Fanuc KAREL source: CA0046.KL

PROGRAM CA0046
%STACKSIZE=65535
%PRIORITY=65535
%NOLOCKGROUP
TYPE
T=STRUCTURE
A : INTEGER
B : REAL
ENDSTRUCTURE
VAR
G : INTEGER
I : INTEGER
R : REAL
B : BOOLEAN
S : STRING[16]
AI : ARRAY[2] OF INTEGER
AR : ARRAY[2] OF REAL
ST : T
P : XYZWPR
V : VECTOR
ROUTINE F(P1 : ARRAY[*] OF INTEGER; P2 : ARRAY[*] OF REAL; P3 : T; P4 : XYZWPR; P5 : VECTOR; P6 : ARRAY[*] OF INTEGER; P7 : ARRAY[*] OF REAL; P8 : T; P9 : XYZWPR; P10 : VECTOR; P11 : ARRAY[*] OF INTEGER;
P12 : ARRAY[*] OF REAL; P13 : T; P14 : XYZWPR; P15 : VECTOR; P16 : ARRAY[*] OF INTEGER; P17 : ARRAY[*] OF REAL; P18 : T; P19 : XYZWPR; P20 : VECTOR; P21 : ARRAY[*] OF INTEGER; P22 : ARRAY[*] OF REAL;
P23 : T; P24 : XYZWPR) FROM CA0046
ROUTINE F
BEGIN
G=(G + 1)
END F
BEGIN
G=0
I=1
R=2.5
B=TRUE
S='A'
AI[1]=3
AR[1]=4.5
-- UNSAFE_SOURCE_IR line 54: ST.A = 5
-- UNSAFE_SOURCE_IR line 55: ST.B = 6.5
F(AI,AR,ST,P,V,AI,AR,ST,P,V,AI,AR,ST,P,V,AI,AR,ST,P,V,AI,AR,ST,P)
END CA0046
